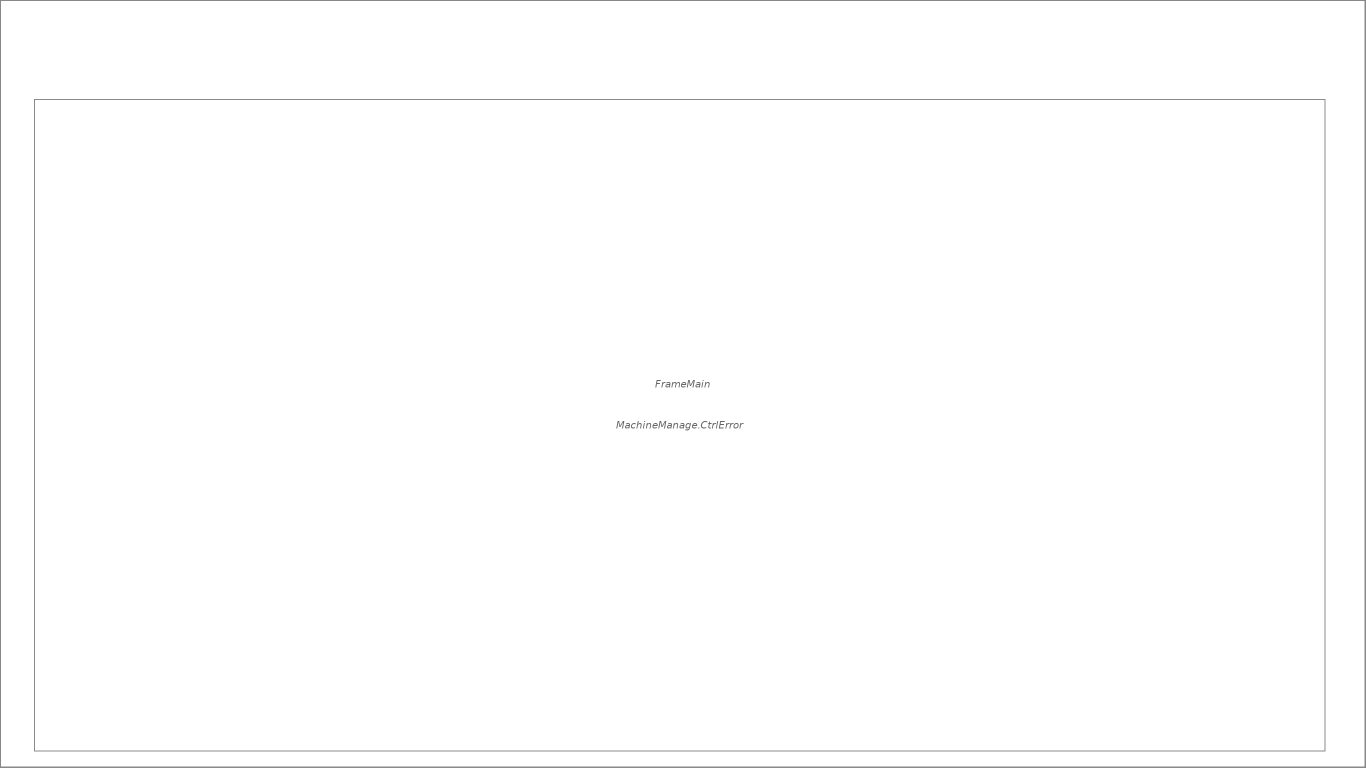
VISUALIZATION PageMessage  // 1366x768
    Frame (0,0 1366x768)
        shows FrameMain()
    Frame (34,99 1291x652)
        shows MachineManage.CtrlError(System := G_stSystem, Error := G_stError)
END_VISUALIZATION

(* stored: Version 1.1.0.1, ProductVersion 3.1.4024.3
   Visu PageMessage: Id {27928c79-8568-45e9-9525-e3cbf24a4ae6} *)
